{attribute 'pack_mode' := '1'}
TYPE ST_AdsCommandBatch :
	STRUCT
		nMagic : UDINT := 16#41434D44;       // "ACMD"
		nFormatVersion : UINT := 4;
		nPayloadSize : UINT := 1888;
		nSequenceStart : UDINT := 0;
		nRequestId : UDINT := 0;
		nAxisMask : BYTE := 0;               // bit0=X, bit1=Y
		bEnsurePower : BOOL := TRUE;
		nReserved : UINT := 0;
		stAxisX : ST_AdsAxisCommand;
		stAxisY : ST_AdsAxisCommand;
		nSequenceEnd : UDINT := 0;
	END_STRUCT
END_TYPE

(* stored: Version 1.1.0.1, ProductVersion 3.1.4024.15
   DUT ST_AdsCommandBatch: Id {0132fd1b-3064-42f1-a003-58f274bd543f} *)
